// TIA Portal V17 export
// export: Created 2023-12-22T15:08:02.4523829Z, ExportSetting WithDefaults, DisplayName Totally Integrated Automation Portal, DisplayVersion V17, DisplayName TIA Portal Openness, DisplayVersion V17, DisplayName TIA Portal Version Control Interface, DisplayVersion V17, DisplayName STEP 7 Professional, DisplayVersion V17, DisplayName STEP 7 Safety, DisplayVersion V17, DisplayName WinCC Advanced, DisplayVersion V17
FUNCTION_BLOCK "Valves"   // FB250, LAD
TITLE = Клапана
{ S7_Optimized_Access := 'FALSE' }
VERSION : 0.1
// FB_Alarm - аварийный сигнал для отключения клапана (например по давлению воздуха), 0 - авария, 1 - норма
// FB_QF - сигнал готовности к работе (например, по наличию 24в в линии управления пневмораспределителем), 0 - авария, 1 - норма
// FB_Open - обратная связь датчика открытия клапана, 0 - закрыт, 1 - открыт
// FB_Close - обратная связь датчика закрытия клапана, 1 - закрыт, 0 - открыт
// Value - управление аналоговым клапаном с позиционированием, формат Real, передаётся в блок AO_ex для конвертации в выходной сигнал контроллера (PQW), для использования установите #CMD.Analog в True
// 
// Q -  постоянный сигнал управления клапаном, 0 - закрыть, 1 - открыть
// stored: AutoNumber false, IsIECCheckEnabled false, SetENOAutomatically false, UDAEnableTagReadback false
   VAR DB_SPECIFIC
      Time_DTL { S7_SetPoint := 'True'} : DTL;
   END_VAR
   VAR_TEMP   // added for the SCL form of the ladder/FBD networks
      _w1 : Bool;
   END_VAR
BEGIN

REGION Network 1: Задвижки
END_REGION

REGION Network 2: Внешняя авария
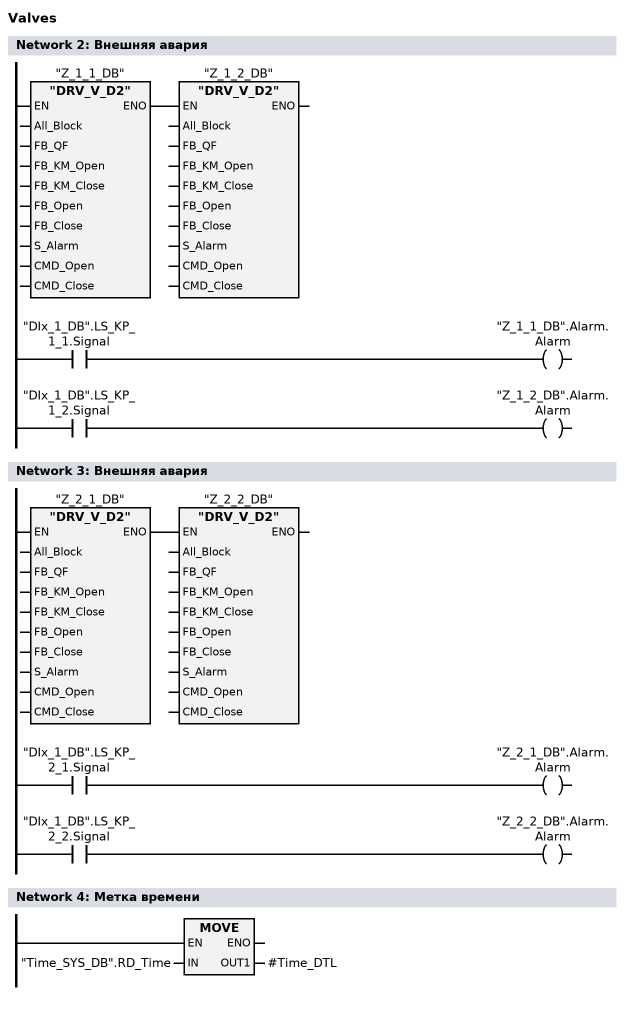
   RUNG wire#powerrail
      "Z_1_1_DB"(All_Block :=, FB_QF :=, FB_KM_Open :=, FB_KM_Close :=, FB_Open :=, FB_Close :=, S_Alarm :=, CMD_Open :=, CMD_Close :=)
      "Z_1_2_DB"(All_Block :=, FB_QF :=, FB_KM_Open :=, FB_KM_Close :=, FB_Open :=, FB_Close :=, S_Alarm :=, CMD_Open :=, CMD_Close :=)
   END_RUNG
   RUNG wire#powerrail
      Contact( "DIx_1_DB".LS_KP_1_1.Signal )
      Coil( "Z_1_1_DB".Alarm.Alarm )
   END_RUNG
   RUNG wire#powerrail
      Contact( "DIx_1_DB".LS_KP_1_2.Signal )
      Coil( "Z_1_2_DB".Alarm.Alarm )
   END_RUNG
   // the same network as SCL:
   "Z_1_1_DB"(ENO => #_w1);   // "DRV_V_D2"
   IF #_w1 THEN
       "Z_1_2_DB"();   // "DRV_V_D2"
   END_IF;
   "Z_1_1_DB".Alarm.Alarm := "DIx_1_DB".LS_KP_1_1.Signal;
   "Z_1_2_DB".Alarm.Alarm := "DIx_1_DB".LS_KP_1_2.Signal;
END_REGION

REGION Network 3: Внешняя авария
   RUNG wire#powerrail
      "Z_2_1_DB"(All_Block :=, FB_QF :=, FB_KM_Open :=, FB_KM_Close :=, FB_Open :=, FB_Close :=, S_Alarm :=, CMD_Open :=, CMD_Close :=)
      "Z_2_2_DB"(All_Block :=, FB_QF :=, FB_KM_Open :=, FB_KM_Close :=, FB_Open :=, FB_Close :=, S_Alarm :=, CMD_Open :=, CMD_Close :=)
   END_RUNG
   RUNG wire#powerrail
      Contact( "DIx_1_DB".LS_KP_2_1.Signal )
      Coil( "Z_2_1_DB".Alarm.Alarm )
   END_RUNG
   RUNG wire#powerrail
      Contact( "DIx_1_DB".LS_KP_2_2.Signal )
      Coil( "Z_2_2_DB".Alarm.Alarm )
   END_RUNG
   // the same network as SCL:
   "Z_2_1_DB"(ENO => #_w1);   // "DRV_V_D2"
   IF #_w1 THEN
       "Z_2_2_DB"();   // "DRV_V_D2"
   END_IF;
   "Z_2_1_DB".Alarm.Alarm := "DIx_1_DB".LS_KP_2_1.Signal;
   "Z_2_2_DB".Alarm.Alarm := "DIx_1_DB".LS_KP_2_2.Signal;
END_REGION

REGION Network 4: Метка времени
   RUNG wire#powerrail
      Move(in := "Time_SYS_DB".RD_Time, out1 => #Time_DTL)
   END_RUNG
   // the same network as SCL:
   #Time_DTL := "Time_SYS_DB".RD_Time;
END_REGION
END_FUNCTION_BLOCK
